{attribute 'qualified_only'}
{attribute 'strict'}
TYPE 
	MotorVenderEnum					: (SANYO, DELTA, YASKAWA);
END_TYPE

(* stored: Version 1.1.0.1, ProductVersion 3.1.4024.9
   DUT MotorVenderEnum: Id {d213547f-5a27-4216-9c67-7c8482aa86bf} *)
